FUNCTION_BLOCK Client (* Basic FB with empty ECC *)
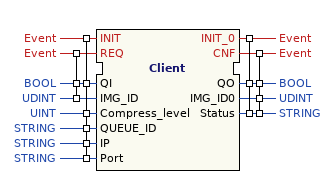
  EVENT_INPUT
    INIT WITH QI, Compress_level, QUEUE_ID, IP, Port;
    REQ WITH QI, IMG_ID;
  END_EVENT
  EVENT_OUTPUT
    INIT_0 WITH Status, QO;
    CNF WITH Status, IMG_ID0, QO;
  END_EVENT
  VAR_INPUT
    QI : BOOL;
    IMG_ID : UDINT;
    Compress_level : UINT;
    QUEUE_ID : STRING;
    IP : STRING;
    Port : STRING;
  END_VAR
  VAR_OUTPUT
    QO : BOOL;
    IMG_ID0 : UDINT;
    Status : STRING;
  END_VAR
END_FUNCTION_BLOCK
